(* CODESYS project TcL_Timers.library
   Company: TwinCAT Libre
   DocFormat: reStructuredText
   Description: Basic timing functions
   Version: 0.1
   Placeholder: TcL_Timers
   Author: Ryan Severson
   Title: TcL_Timers

Project tree, tasks and I/O mapping:
  libraries: Tc2_Standard, * (Beckhoff Automation GmbH)
  imgs/
    Heartbeat.jpg
    TOF.jpg
    TOFRT.jpg
    TON.jpg
    TONRT.jpg
    Watchdog.jpg
  00000000-0000-0000-0000-000000000000|imgs\Heartbeat.jpg
  00000000-0000-0000-0000-000000000000|imgs\TOF.jpg
  00000000-0000-0000-0000-000000000000|imgs\TOFRT.jpg
  00000000-0000-0000-0000-000000000000|imgs\TON.jpg
  00000000-0000-0000-0000-000000000000|imgs\TONRT.jpg
  00000000-0000-0000-0000-000000000000|imgs\Watchdog.jpg
  Project Information/
    function F_GetCompany [ST]
    function F_GetTitle [ST]
    function F_GetVersion [ST]
  Version/
    global variables Global_Version
  function block fb_BaseTimer [ST]
  function block fb_Heartbeat [ST]
  function block fb_TOF [ST]
  function block fb_TOFRT [ST]
  function block fb_TON [ST]
  function block fb_TONRT [ST]
  function block fb_Watchdog [ST]
*)

// Version/Global_Version
{attribute 'TcGenerated'}
{attribute 'no-analysis'}
{attribute 'linkalways'}
// This function has been automatically generated from the project information.
VAR_GLOBAL CONSTANT
	{attribute 'const_non_replaced'}
	stLibVersion_TcL_Timers : ST_LibVersion := (iMajor := 0, iMinor := 1, iBuild := 0, iRevision := 0, nFlags := 0, sVersion := '0.1');
END_VAR

// Project Information/F_GetCompany
// This function has been automatically generated from the project information.
{attribute 'signature_flag' := '1073741824'}
{attribute 'TcGenerated'}
{attribute 'no-analysis'}
FUNCTION F_GetCompany : WSTRING
VAR_INPUT
	
END_VAR

F_GetCompany := "TwinCAT Libre";

END_FUNCTION

// Project Information/F_GetTitle
// This function has been automatically generated from the project information.
{attribute 'signature_flag' := '1073741824'}
{attribute 'TcGenerated'}
{attribute 'no-analysis'}
FUNCTION F_GetTitle : WSTRING
VAR_INPUT
	
END_VAR

F_GetTitle := "TcL_Timers";

END_FUNCTION

// Project Information/F_GetVersion
// This function has been automatically generated from the project information.
{attribute 'signature_flag' := '1073741824'}
{attribute 'TcGenerated'}
{attribute 'no-analysis'}
FUNCTION F_GetVersion : ST_LibVersion
VAR_INPUT
	
END_VAR

F_GetVersion.iMajor := 0;
F_GetVersion.iMinor := 1;
F_GetVersion.iBuild := 0;
F_GetVersion.iRevision := 0;

END_FUNCTION

// fb_BaseTimer
(*
:Info: https://github.com/TwinCAT-Libre/
:Author: TwinCAT Libre

Version history:

+-------------+------------+----------+------------------------------------------+
|Date         | Version    | Author   | Remark                                   |
+=============+============+==========+==========================================+
|2022-03-20   | 0.1        | R.S.     | Initial Release                          |
+-------------+------------+----------+------------------------------------------+

*)

{attribute 'conditionalshow'}
FUNCTION_BLOCK fb_BaseTimer
//Base fb for all TON, TOF and their extensions
VAR_INPUT
	PT : TIME := T#0S; //Preset Time
END_VAR
VAR_OUTPUT
	RT : TIME := T#0S; //Remaining Time
	ET : TIME := T#0S; //Elapsed Time
	{attribute 'dataflow'}
	Q : BOOL := FALSE;  //Output
	TT : BOOL := FALSE; //Timer is Timing (active)
END_VAR
VAR
END_VAR

END_FUNCTION_BLOCK

// fb_Heartbeat
(*
:Info: https://github.com/TwinCAT-Libre/
:Author: TwinCAT Libre

Version history:

+-------------+------------+----------+------------------------------------------+
|Date         | Version    | Author   | Remark                                   |
+=============+============+==========+==========================================+
|2022-03-20   | 0.1        | R.S.     | Initial Release                          |
+-------------+------------+----------+------------------------------------------+

Timing Diagram: 

.. image:: ../imgs/Heartbeat.jpg

*)

{attribute 'hide_all_locals'}
{attribute 'conditionalshow_all_locals'}
FUNCTION_BLOCK fb_Heartbeat
//Generates a toggling signal to be monitored externally
//Q toggles one cycle in FT  
VAR_INPUT
	Enable : BOOL := TRUE;//Allow the heartbeat to occur 
	FT : TIME := T#5S;//Period of heartbeat
END_VAR
VAR_OUTPUT
	Q : BOOL :=FALSE; //Heartbeat
END_VAR
VAR
	_tpOn : TP;
	_tpOff : TP;
END_VAR

_tpOn(IN:= Enable AND NOT _tpOff.q,PT:=FT/2, Q=>Q);
_tpOff(IN:= Enable AND NOT _tpOn.Q,PT:=FT/2);

END_FUNCTION_BLOCK

// fb_TOF
(*
:Info: https://github.com/TwinCAT-Libre/
:Author: TwinCAT Libre

Version history:

+-------------+------------+----------+------------------------------------------+
|Date         | Version    | Author   | Remark                                   |
+=============+============+==========+==========================================+
|2022-03-20   | 0.1        | R.S.     | Initial Release                          |
+-------------+------------+----------+------------------------------------------+

Timing Diagram: 

.. image:: ../imgs/TOF.jpg
*)

FUNCTION_BLOCK fb_TOF EXTENDS fb_BaseTimer
//Basic timer with additional functionality, drop in replacement for basic TOF
VAR_INPUT
	{attribute 'dataflow'}
	IN : BOOL :=TRUE;
END_VAR
VAR
	_tof : TOF; //Internal base timer reference
END_VAR

//instantiation
_tof(IN:=IN,PT:=PT,Q=>Q,ET=>ET);
 
//set/evaluate outputs
TT := (NOT _tof.IN AND _tof.Q);
RT := _tof.PT - _tof.ET;

END_FUNCTION_BLOCK

// fb_TOFRT
(*
:Info: https://github.com/TwinCAT-Libre/
:Author: TwinCAT Libre

Version history:

+-------------+------------+----------+------------------------------------------+
|Date         | Version    | Author   | Remark                                   |
+=============+============+==========+==========================================+
|2022-03-20   | 0.1        | R.S.     | Initial Release                          |
+-------------+------------+----------+------------------------------------------+

Timing Diagram: 

.. image:: ../imgs/TOFRT.jpg
*)

{attribute 'hide_all_locals'}
{attribute 'conditionalshow_all_locals'}
FUNCTION_BLOCK fb_TOFRT EXTENDS fb_TOF
//Time off delay - Retentive. Accumulates time until complete or reset
//Clearing IN after timer completes will reset the timer
VAR_INPUT
	Reset : BOOL :=FALSE; //Set TRUE to restart the timer, either when running, done or paused
END_VAR
VAR_OUTPUT
	Paused :BOOL:=FALSE; //Timer paused
END_VAR
VAR 
	_pausedTime : TIME := T#0S; //holder for pause state
	_elapsedTime : TIME := T#0S; //holder for elapsed time
	_osr : R_TRIG;
	_osf : F_TRIG;
END_VAR

//start detection
_osf(CLK:=IN);
IF _osf.q AND Paused AND Q THEN //resume case
	_tof.PT:=_pausedTime;
	Paused:=FALSE;
	ELSIF _osf.q AND _pausedTime=T#0S THEN //start case
	_tof.PT:=PT;
	ELSIF _osf.q AND NOT Q THEN //restart case after completion
	_tof.PT:=PT;
	Paused:=FALSE;	
END_IF

//stop detection
_osr(CLK:=IN);
IF _osr.q AND Q THEN //regular pause case
	_pausedTime := _tof.PT - _tof.ET;
	_elapsedTime := _tof.ET + _elapsedTime;	
	Paused:=TRUE;
	ELSIF _osr.q AND NOT Q THEN //restart case
	_pausedTime := T#0S;
	_elapsedTime := T#0S;
	_tof.PT := T#0S;
END_IF

//reset handling
IF Reset THEN
	_pausedTime := T#0S;
	_elapsedTime := T#0S;
	_tof.PT := PT;
	Paused :=FALSE;
END_IF


//timer call
//_tof(IN:=(IN AND NOT RESET),Q=>Q);
IF RESET THEN
		_tof(IN:=TRUE,Q=>Q);
	ELSE
		_tof(IN:=(IN),Q=>Q);
END_IF

//purely aesthetic
IF Paused THEN
	RT:= _pausedTime;
	ET:=_elapsedTime;
	ELSE
	RT:=_tof.PT-_tof.ET;	
	ET:=_tof.ET + _elapsedTime;	
END_IF

TT := (NOT _tof.IN AND _tof.Q);

END_FUNCTION_BLOCK

// fb_TON
(*
:Info: https://github.com/TwinCAT-Libre/
:Author: TwinCAT Libre

Version history:

+-------------+------------+----------+------------------------------------------+
|Date         | Version    | Author   | Remark                                   |
+=============+============+==========+==========================================+
|2022-03-20   | 0.1        | R.S.     | Initial Release                          |
+-------------+------------+----------+------------------------------------------+

.. image:: ../imgs/TON.jpg
*)

{attribute 'hide_all_locals'}
{attribute 'conditionalshow_all_locals'}
FUNCTION_BLOCK fb_TON EXTENDS fb_BaseTimer
//Basic timer with additional functionality, drop in replacement for basic TON
VAR_INPUT
	{attribute 'dataflow'}
	IN : BOOL :=FALSE;
END_VAR

VAR
	_ton : TON; //Internal base timer reference
END_VAR

//instantiation
_ton(IN:=IN,PT:=PT,Q=>Q,ET=>ET);
 
//set/evaluate outputs
TT := (_ton.IN AND NOT _ton.Q);
RT := _ton.PT - _ton.ET;

END_FUNCTION_BLOCK

// fb_TONRT
(*
:Info: https://github.com/TwinCAT-Libre/
:Author: TwinCAT Libre

Version history:

+-------------+------------+----------+------------------------------------------+
|Date         | Version    | Author   | Remark                                   |
+=============+============+==========+==========================================+
|2022-03-20   | 0.1        | R.S.     | Initial Release                          |
+-------------+------------+----------+------------------------------------------+

Timing Diagram: 

.. image:: ../imgs/TONRT.jpg
*)

{attribute 'hide_all_locals'}
{attribute 'conditionalshow_all_locals'}
FUNCTION_BLOCK fb_TONRT EXTENDS fb_TON
//Time on delay - Retentive. Accumulates time until complete or reset
//Clearing IN after timer completes will reset the timer
VAR_INPUT
	Reset : BOOL :=FALSE; //Set TRUE to restart the timer, either when running, done or paused
END_VAR
VAR_OUTPUT
	Paused :BOOL:=FALSE; //Timer paused
END_VAR
VAR 
	_pausedTime : TIME := T#0S; //holder for pause state
	_elapsedTime : TIME := T#0S; //holder for elapsed time
	_osr : R_TRIG;
	_osf : F_TRIG;
END_VAR

//start detection
_osr(CLK:=IN);
IF _osr.q AND Paused AND NOT Q THEN //resume case
	_ton.PT:=_pausedTime;
	Paused:=FALSE;
	ELSIF _osr.q AND _pausedTime=T#0S THEN //start case
	_ton.PT:=PT;
	ELSIF _osr.q AND Q THEN //restart case after completion
	_ton.PT:=PT;
	Paused:=FALSE;	
END_IF

//stop detection
_osf(CLK:=IN);
IF _osf.q AND NOT Q THEN //regular pause case
	_pausedTime := _ton.PT - _ton.ET;
	_elapsedTime := _ton.ET + _elapsedTime;	
	Paused:=TRUE;
	ELSIF _osf.q AND Q THEN //restart case
	_pausedTime := T#0S;
	_elapsedTime := T#0S;
	_ton.PT := T#0S;
END_IF

//reset handling
IF Reset THEN
	_pausedTime := T#0S;
	_elapsedTime := T#0S;
	_ton.PT := PT;
	Paused :=FALSE;
END_IF


//timer call
_ton(IN:=(IN AND NOT RESET),Q=>Q);

//purely aesthetic
IF Paused THEN
	RT:= _pausedTime;
	ET:=_elapsedTime;
	ELSE
	RT:=_ton.PT-_ton.ET;	
	ET:=_ton.ET + _elapsedTime;
END_IF


TT := (_ton.IN AND NOT _ton.Q);

END_FUNCTION_BLOCK

// fb_Watchdog
(*
:Info: https://github.com/TwinCAT-Libre/
:Author: TwinCAT Libre

Version history:

+-------------+------------+----------+------------------------------------------+
|Date         | Version    | Author   | Remark                                   |
+=============+============+==========+==========================================+
|2022-03-20   | 0.1        | R.S.     | Initial Release                          |
+-------------+------------+----------+------------------------------------------+

Timing Diagram: 

.. image:: ../imgs/Watchdog.jpg
*)

{attribute 'hide_all_locals'}
{attribute 'conditionalshow_all_locals'}
FUNCTION_BLOCK fb_Watchdog
//Monitors an external toggling signal
//Sets alarm if no change occurs in SIGNAL in the timeout period
VAR_INPUT
	{attribute 'dataflow'}
	Enable : BOOL := TRUE; //Enables the evaluation 
	Timeout : TIME := T#5S; //If signal is stale for this time, set the alarm
	Signal : BOOL :=FALSE; //Signal to monitor
END_VAR
VAR_OUTPUT
	{attribute 'dataflow'}
	Alarm : BOOL :=FALSE;
END_VAR
VAR
	_ton : TON;
	_osr : R_TRIG;
	_osf : F_TRIG;
END_VAR

_osr(CLK:=Signal);
_osf(CLK:=Signal);

_ton(IN:=Enable AND (NOT _osr.q) AND (NOT _osf.q),PT:=Timeout, Q=>Alarm);

END_FUNCTION_BLOCK
